(* IEC 61131-3 sources: mect_apps/TPAC1008_02_AF/Octopus_Prey/plc, 2 files *)

(* ---- Crosstable.gvl ---- *)
VAR_GLOBAL
	STATUS AT %QW0.772:UINT;
	RTU_HEARTBEAT AT %IW0.800:UINT;
	RTU_RTU_WR AT %QX0.804.0:BOOL;
	RTU_RTU_RD AT %IX0.808.0:BOOL;
	TEST_COMMAND AT %IW0.15896:UINT;
	TST_DigIn_1 AT %IX0.15900.0:BOOL;
	TST_DigIn_2 AT %IX0.15904.0:BOOL;
	TST_DigIn_3 AT %IX0.15908.0:BOOL;
	TST_DigIn_4 AT %IX0.15912.0:BOOL;
	TST_DigIn_5 AT %IX0.15916.0:BOOL;
	TST_DigIn_6 AT %IX0.15920.0:BOOL;
	TST_DigIn_7 AT %IX0.15924.0:BOOL;
	TST_DigIn_8 AT %IX0.15928.0:BOOL;
	TST_DigIn_9 AT %IX0.15932.0:BOOL;
	TST_DigIn_10 AT %IX0.15936.0:BOOL;
	TST_DigIn_11 AT %IX0.15940.0:BOOL;
	TST_DigIn_12 AT %IX0.15944.0:BOOL;
	TST_DigIn_13 AT %IX0.15948.0:BOOL;
	TST_DigIn_14 AT %IX0.15952.0:BOOL;
	TST_DigIn_15 AT %IX0.15956.0:BOOL;
	TST_DigIn_16 AT %IX0.15960.0:BOOL;
	VAL_DigIn_1 AT %IX0.15964.0:BOOL;
	VAL_DigIn_2 AT %IX0.15968.0:BOOL;
	VAL_DigIn_3 AT %IX0.15972.0:BOOL;
	VAL_DigIn_4 AT %IX0.15976.0:BOOL;
	VAL_DigIn_5 AT %IX0.15980.0:BOOL;
	VAL_DigIn_6 AT %IX0.15984.0:BOOL;
	VAL_DigIn_7 AT %IX0.15988.0:BOOL;
	VAL_DigIn_8 AT %IX0.15992.0:BOOL;
	VAL_DigIn_9 AT %IX0.15996.0:BOOL;
	VAL_DigIn_10 AT %IX0.16000.0:BOOL;
	VAL_DigIn_11 AT %IX0.16004.0:BOOL;
	VAL_DigIn_12 AT %IX0.16008.0:BOOL;
	VAL_DigIn_13 AT %IX0.16012.0:BOOL;
	VAL_DigIn_14 AT %IX0.16016.0:BOOL;
	VAL_DigIn_15 AT %IX0.16020.0:BOOL;
	VAL_DigIn_16 AT %IX0.16024.0:BOOL;
	RES_DigIn_1 AT %QX0.16028.0:BOOL;
	RES_DigIn_2 AT %QX0.16032.0:BOOL;
	RES_DigIn_3 AT %QX0.16036.0:BOOL;
	RES_DigIn_4 AT %QX0.16040.0:BOOL;
	RES_DigIn_5 AT %QX0.16044.0:BOOL;
	RES_DigIn_6 AT %QX0.16048.0:BOOL;
	RES_DigIn_7 AT %QX0.16052.0:BOOL;
	RES_DigIn_8 AT %QX0.16056.0:BOOL;
	RES_DigIn_9 AT %QX0.16060.0:BOOL;
	RES_DigIn_10 AT %QX0.16064.0:BOOL;
	RES_DigIn_11 AT %QX0.16068.0:BOOL;
	RES_DigIn_12 AT %QX0.16072.0:BOOL;
	RES_DigIn_13 AT %QX0.16076.0:BOOL;
	RES_DigIn_14 AT %QX0.16080.0:BOOL;
	RES_DigIn_15 AT %QX0.16084.0:BOOL;
	RES_DigIn_16 AT %QX0.16088.0:BOOL;
	TST_DigOut_1 AT %IX0.16092.0:BOOL;
	TST_DigOut_2 AT %IX0.16096.0:BOOL;
	TST_DigOut_3 AT %IX0.16100.0:BOOL;
	TST_DigOut_4 AT %IX0.16104.0:BOOL;
	TST_DigOut_5 AT %IX0.16108.0:BOOL;
	TST_DigOut_6 AT %IX0.16112.0:BOOL;
	TST_DigOut_7 AT %IX0.16116.0:BOOL;
	TST_DigOut_8 AT %IX0.16120.0:BOOL;
	TST_DigOut_9 AT %IX0.16124.0:BOOL;
	TST_DigOut_10 AT %IX0.16128.0:BOOL;
	TST_DigOut_11 AT %IX0.16132.0:BOOL;
	TST_DigOut_12 AT %IX0.16136.0:BOOL;
	TST_DigOut_13 AT %IX0.16140.0:BOOL;
	TST_DigOut_14 AT %IX0.16144.0:BOOL;
	TST_DigOut_15 AT %IX0.16148.0:BOOL;
	TST_DigOut_16 AT %IX0.16152.0:BOOL;
	VAL_DigOut_1 AT %IX0.16156.0:BOOL;
	VAL_DigOut_2 AT %IX0.16160.0:BOOL;
	VAL_DigOut_3 AT %IX0.16164.0:BOOL;
	VAL_DigOut_4 AT %IX0.16168.0:BOOL;
	VAL_DigOut_5 AT %IX0.16172.0:BOOL;
	VAL_DigOut_6 AT %IX0.16176.0:BOOL;
	VAL_DigOut_7 AT %IX0.16180.0:BOOL;
	VAL_DigOut_8 AT %IX0.16184.0:BOOL;
	VAL_DigOut_9 AT %IX0.16188.0:BOOL;
	VAL_DigOut_10 AT %IX0.16192.0:BOOL;
	VAL_DigOut_11 AT %IX0.16196.0:BOOL;
	VAL_DigOut_12 AT %IX0.16200.0:BOOL;
	VAL_DigOut_13 AT %IX0.16204.0:BOOL;
	VAL_DigOut_14 AT %IX0.16208.0:BOOL;
	VAL_DigOut_15 AT %IX0.16212.0:BOOL;
	VAL_DigOut_16 AT %IX0.16216.0:BOOL;
	TST_AnIn_1 AT %IX0.16220.0:BOOL;
	TST_AnIn_2 AT %IX0.16224.0:BOOL;
	TST_AnIn_3 AT %IX0.16228.0:BOOL;
	TST_AnIn_4 AT %IX0.16232.0:BOOL;
	TST_AnIn_5 AT %IX0.16236.0:BOOL;
	TST_AnIn_6 AT %IX0.16240.0:BOOL;
	TST_AnIn_7 AT %IX0.16244.0:BOOL;
	TST_AnIn_8 AT %IX0.16248.0:BOOL;
	TST_AnIn_9 AT %IX0.16252.0:BOOL;
	TST_AnIn_10 AT %IX0.16256.0:BOOL;
	TST_AnIn_11 AT %IX0.16260.0:BOOL;
	TST_AnIn_12 AT %IX0.16264.0:BOOL;
	VAL_AnIn_1 AT %IW0.16268:INT;
	VAL_AnIn_2 AT %IW0.16272:INT;
	VAL_AnIn_3 AT %IW0.16276:INT;
	VAL_AnIn_4 AT %IW0.16280:INT;
	VAL_AnIn_5 AT %IW0.16284:INT;
	VAL_AnIn_6 AT %IW0.16288:INT;
	VAL_AnIn_7 AT %IW0.16292:INT;
	VAL_AnIn_8 AT %IW0.16296:INT;
	VAL_AnIn_9 AT %IW0.16300:INT;
	VAL_AnIn_10 AT %IW0.16304:INT;
	VAL_AnIn_11 AT %IW0.16308:INT;
	VAL_AnIn_12 AT %IW0.16312:INT;
	VAL_AnInConf_1 AT %IW0.16316:UINT;
	VAL_AnInConf_2 AT %IW0.16320:UINT;
	VAL_AnInConf_3 AT %IW0.16324:UINT;
	VAL_AnInConf_4 AT %IW0.16328:UINT;
	VAL_AnInConf_5 AT %IW0.16332:UINT;
	VAL_AnInConf_6 AT %IW0.16336:UINT;
	VAL_AnInConf_7 AT %IW0.16340:UINT;
	VAL_AnInConf_8 AT %IW0.16344:UINT;
	VAL_AnInConf_9 AT %IW0.16348:UINT;
	VAL_AnInConf_10 AT %IW0.16352:UINT;
	VAL_AnInConf_11 AT %IW0.16356:UINT;
	VAL_AnInConf_12 AT %IW0.16360:UINT;
	VAL_AnInFltr_1 AT %IW0.16364:UINT;
	VAL_AnInFltr_2 AT %IW0.16368:UINT;
	VAL_AnInFltr_3 AT %IW0.16372:UINT;
	VAL_AnInFltr_4 AT %IW0.16376:UINT;
	VAL_AnInFltr_5 AT %IW0.16380:UINT;
	VAL_AnInFltr_6 AT %IW0.16384:UINT;
	VAL_AnInFltr_7 AT %IW0.16388:UINT;
	VAL_AnInFltr_8 AT %IW0.16392:UINT;
	VAL_AnInFltr_9 AT %IW0.16396:UINT;
	VAL_AnInFltr_10 AT %IW0.16400:UINT;
	VAL_AnInFltr_11 AT %IW0.16404:UINT;
	VAL_AnInFltr_12 AT %IW0.16408:UINT;
	RES_AnIn_1 AT %QW0.16412:INT;
	RES_AnIn_2 AT %QW0.16416:INT;
	RES_AnIn_3 AT %QW0.16420:INT;
	RES_AnIn_4 AT %QW0.16424:INT;
	RES_AnIn_5 AT %QW0.16428:INT;
	RES_AnIn_6 AT %QW0.16432:INT;
	RES_AnIn_7 AT %QW0.16436:INT;
	RES_AnIn_8 AT %QW0.16440:INT;
	RES_AnIn_9 AT %QW0.16444:INT;
	RES_AnIn_10 AT %QW0.16448:INT;
	RES_AnIn_11 AT %QW0.16452:INT;
	RES_AnIn_12 AT %QW0.16456:INT;
	RES_AnInStts_1 AT %QW0.16460:INT;
	RES_AnInStts_2 AT %QW0.16464:INT;
	RES_AnInStts_3 AT %QW0.16468:INT;
	RES_AnInStts_4 AT %QW0.16472:INT;
	RES_AnInStts_5 AT %QW0.16476:INT;
	RES_AnInStts_6 AT %QW0.16480:INT;
	RES_AnInStts_7 AT %QW0.16484:INT;
	RES_AnInStts_8 AT %QW0.16488:INT;
	RES_AnInStts_9 AT %QW0.16492:INT;
	RES_AnInStts_10 AT %QW0.16496:INT;
	RES_AnInStts_11 AT %QW0.16500:INT;
	RES_AnInStts_12 AT %QW0.16504:INT;
	TST_AnOut_1 AT %IX0.16508.0:BOOL;
	TST_AnOut_2 AT %IX0.16512.0:BOOL;
	TST_AnOut_3 AT %IX0.16516.0:BOOL;
	TST_AnOut_4 AT %IX0.16520.0:BOOL;
	VAL_AnOut_1 AT %IW0.16524:INT;
	VAL_AnOut_2 AT %IW0.16528:INT;
	VAL_AnOut_3 AT %IW0.16532:INT;
	VAL_AnOut_4 AT %IW0.16536:INT;
	VAL_AnOutConf_1 AT %IW0.16540:UINT;
	VAL_AnOutConf_2 AT %IW0.16544:UINT;
	VAL_AnOutConf_3 AT %IW0.16548:UINT;
	VAL_AnOutConf_4 AT %IW0.16552:UINT;
	RES_AnOutStts_1 AT %QW0.16556:INT;
	RES_AnOutStts_2 AT %QW0.16560:INT;
	RES_AnOutStts_3 AT %QW0.16564:INT;
	RES_AnOutStts_4 AT %QW0.16568:INT;
	TST_Tamb AT %IX0.16572.0:BOOL;
	TST_RPM AT %IX0.16576.0:BOOL;
	TST_FWrevision AT %IX0.16580.0:BOOL;
	TST_HWconfig AT %IX0.16584.0:BOOL;
	VAL_Tamb AT %IW0.16588:INT;
	VAL_RPM AT %IW0.16592:UINT;
	VAL_FWrevision AT %IW0.16596:UINT;
	VAL_HWconfig AT %IW0.16600:UINT;
	RES_Tamb AT %QW0.16604:INT;
	RES_RPM AT %QW0.16608:UINT;
	RES_FWrevision AT %QW0.16612:UINT;
	RES_HWconfig AT %QW0.16616:UINT;
	TST_RTUS_WR AT %IX0.16620.0:BOOL;
	TST_RTUS_RD AT %IX0.16624.0:BOOL;
	TST_RTU1_WR AT %IX0.16628.0:BOOL;
	TST_RTU1_RD AT %IX0.16632.0:BOOL;
	TST_RTU3_WR AT %IX0.16636.0:BOOL;
	TST_RTU3_RD AT %IX0.16640.0:BOOL;
	TST_CAN1_WR AT %IX0.16644.0:BOOL;
	TST_CAN1_RD AT %IX0.16648.0:BOOL;
	VAL_RTUS_WR AT %IX0.16652.0:BOOL;
	VAL_RTUS_RD AT %IX0.16656.0:BOOL;
	VAL_RTU1_WR AT %IX0.16660.0:BOOL;
	VAL_RTU1_RD AT %IX0.16664.0:BOOL;
	VAL_RTU3_WR AT %IX0.16668.0:BOOL;
	VAL_RTU3_RD AT %IX0.16672.0:BOOL;
	VAL_CAN1_WR AT %IX0.16676.0:BOOL;
	VAL_CAN1_RD AT %IX0.16680.0:BOOL;
	RES_RTUS_WR AT %QX0.16684.0:BOOL;
	RES_RTUS_RD AT %QX0.16688.0:BOOL;
	RES_RTU1_WR AT %QX0.16692.0:BOOL;
	RES_RTU1_RD AT %QX0.16696.0:BOOL;
	RES_RTU3_WR AT %QX0.16700.0:BOOL;
	RES_RTU3_RD AT %QX0.16704.0:BOOL;
	RES_CAN1_WR AT %QX0.16708.0:BOOL;
	RES_CAN1_RD AT %QX0.16712.0:BOOL;
	TEST_STATUS AT %QW0.16716:UINT;
	RTU0_TYPE_PORT AT %ID0.20000:UDINT;
	RTU0_BAUDRATE AT %ID0.20004:UDINT;
	RTU0_STATUS AT %ID0.20008:UDINT;
	RTU0_READS AT %ID0.20012:UDINT;
	RTU0_WRITES AT %ID0.20016:UDINT;
	RTU0_TIMEOUTS AT %ID0.20020:UDINT;
	RTU0_COMM_ERRORS AT %ID0.20024:UDINT;
	RTU0_LAST_ERROR AT %ID0.20028:UDINT;
	RTU0_WRITE_QUEUE AT %ID0.20032:UDINT;
	RTU0_BUS_LOAD AT %ID0.20036:UDINT;
	RTU1_TYPE_PORT AT %ID0.20040:UDINT;
	RTU1_BAUDRATE AT %ID0.20044:UDINT;
	RTU1_STATUS AT %ID0.20048:UDINT;
	RTU1_READS AT %ID0.20052:UDINT;
	RTU1_WRITES AT %ID0.20056:UDINT;
	RTU1_TIMEOUTS AT %ID0.20060:UDINT;
	RTU1_COMM_ERRORS AT %ID0.20064:UDINT;
	RTU1_LAST_ERROR AT %ID0.20068:UDINT;
	RTU1_WRITE_QUEUE AT %ID0.20072:UDINT;
	RTU1_BUS_LOAD AT %ID0.20076:UDINT;
	RTU3_TYPE_PORT AT %ID0.20080:UDINT;
	RTU3_BAUDRATE AT %ID0.20084:UDINT;
	RTU3_STATUS AT %ID0.20088:UDINT;
	RTU3_READS AT %ID0.20092:UDINT;
	RTU3_WRITES AT %ID0.20096:UDINT;
	RTU3_TIMEOUTS AT %ID0.20100:UDINT;
	RTU3_COMM_ERRORS AT %ID0.20104:UDINT;
	RTU3_LAST_ERROR AT %ID0.20108:UDINT;
	RTU3_WRITE_QUEUE AT %ID0.20112:UDINT;
	RTU3_BUS_LOAD AT %ID0.20116:UDINT;
	CAN0_TYPE_PORT AT %ID0.20120:UDINT;
	CAN0_BAUDRATE AT %ID0.20124:UDINT;
	CAN0_STATUS AT %ID0.20128:UDINT;
	CAN0_READS AT %ID0.20132:UDINT;
	CAN0_WRITES AT %ID0.20136:UDINT;
	CAN0_TIMEOUTS AT %ID0.20140:UDINT;
	CAN0_COMM_ERRORS AT %ID0.20144:UDINT;
	CAN0_LAST_ERROR AT %ID0.20148:UDINT;
	CAN0_WRITE_QUEUE AT %ID0.20152:UDINT;
	CAN0_BUS_LOAD AT %ID0.20156:UDINT;
	CAN1_TYPE_PORT AT %ID0.20160:UDINT;
	CAN1_BAUDRATE AT %ID0.20164:UDINT;
	CAN1_STATUS AT %ID0.20168:UDINT;
	CAN1_READS AT %ID0.20172:UDINT;
	CAN1_WRITES AT %ID0.20176:UDINT;
	CAN1_TIMEOUTS AT %ID0.20180:UDINT;
	CAN1_COMM_ERRORS AT %ID0.20184:UDINT;
	CAN1_LAST_ERROR AT %ID0.20188:UDINT;
	CAN1_WRITE_QUEUE AT %ID0.20192:UDINT;
	CAN1_BUS_LOAD AT %ID0.20196:UDINT;
	TCPS_TYPE_PORT AT %ID0.20200:UDINT;
	TCPS_IP_ADDRESS AT %ID0.20204:UDINT;
	TCPS_STATUS AT %ID0.20208:UDINT;
	TCPS_READS AT %ID0.20212:UDINT;
	TCPS_WRITES AT %ID0.20216:UDINT;
	TCPS_TIMEOUTS AT %ID0.20220:UDINT;
	TCPS_COMM_ERRORS AT %ID0.20224:UDINT;
	TCPS_LAST_ERROR AT %ID0.20228:UDINT;
	TCPS_WRITE_QUEUE AT %ID0.20232:UDINT;
	TCPS_BUS_LOAD AT %ID0.20236:UDINT;
	TCP0_TYPE_PORT AT %ID0.20240:UDINT;
	TCP0_IP_ADDRESS AT %ID0.20244:UDINT;
	TCP0_STATUS AT %ID0.20248:UDINT;
	TCP0_READS AT %ID0.20252:UDINT;
	TCP0_WRITES AT %ID0.20256:UDINT;
	TCP0_TIMEOUTS AT %ID0.20260:UDINT;
	TCP0_COMM_ERRORS AT %ID0.20264:UDINT;
	TCP0_LAST_ERROR AT %ID0.20268:UDINT;
	TCP0_WRITE_QUEUE AT %ID0.20272:UDINT;
	TCP0_BUS_LOAD AT %ID0.20276:UDINT;
	TCP1_TYPE_PORT AT %ID0.20280:UDINT;
	TCP1_IP_ADDRESS AT %ID0.20284:UDINT;
	TCP1_STATUS AT %ID0.20288:UDINT;
	TCP1_READS AT %ID0.20292:UDINT;
	TCP1_WRITES AT %ID0.20296:UDINT;
	TCP1_TIMEOUTS AT %ID0.20300:UDINT;
	TCP1_COMM_ERRORS AT %ID0.20304:UDINT;
	TCP1_LAST_ERROR AT %ID0.20308:UDINT;
	TCP1_WRITE_QUEUE AT %ID0.20312:UDINT;
	TCP1_BUS_LOAD AT %ID0.20316:UDINT;
	TCP2_TYPE_PORT AT %ID0.20320:UDINT;
	TCP2_IP_ADDRESS AT %ID0.20324:UDINT;
	TCP2_STATUS AT %ID0.20328:UDINT;
	TCP2_READS AT %ID0.20332:UDINT;
	TCP2_WRITES AT %ID0.20336:UDINT;
	TCP2_TIMEOUTS AT %ID0.20340:UDINT;
	TCP2_COMM_ERRORS AT %ID0.20344:UDINT;
	TCP2_LAST_ERROR AT %ID0.20348:UDINT;
	TCP2_WRITE_QUEUE AT %ID0.20352:UDINT;
	TCP2_BUS_LOAD AT %ID0.20356:UDINT;
	TCP3_TYPE_PORT AT %ID0.20360:UDINT;
	TCP3_IP_ADDRESS AT %ID0.20364:UDINT;
	TCP3_STATUS AT %ID0.20368:UDINT;
	TCP3_READS AT %ID0.20372:UDINT;
	TCP3_WRITES AT %ID0.20376:UDINT;
	TCP3_TIMEOUTS AT %ID0.20380:UDINT;
	TCP3_COMM_ERRORS AT %ID0.20384:UDINT;
	TCP3_LAST_ERROR AT %ID0.20388:UDINT;
	TCP3_WRITE_QUEUE AT %ID0.20392:UDINT;
	TCP3_BUS_LOAD AT %ID0.20396:UDINT;
	TCP4_TYPE_PORT AT %ID0.20400:UDINT;
	TCP4_IP_ADDRESS AT %ID0.20404:UDINT;
	TCP4_STATUS AT %ID0.20408:UDINT;
	TCP4_READS AT %ID0.20412:UDINT;
	TCP4_WRITES AT %ID0.20416:UDINT;
	TCP4_TIMEOUTS AT %ID0.20420:UDINT;
	TCP4_COMM_ERRORS AT %ID0.20424:UDINT;
	TCP4_LAST_ERROR AT %ID0.20428:UDINT;
	TCP4_WRITE_QUEUE AT %ID0.20432:UDINT;
	TCP4_BUS_LOAD AT %ID0.20436:UDINT;
	TCP5_TYPE_PORT AT %ID0.20440:UDINT;
	TCP5_IP_ADDRESS AT %ID0.20444:UDINT;
	TCP5_STATUS AT %ID0.20448:UDINT;
	TCP5_READS AT %ID0.20452:UDINT;
	TCP5_WRITES AT %ID0.20456:UDINT;
	TCP5_TIMEOUTS AT %ID0.20460:UDINT;
	TCP5_COMM_ERRORS AT %ID0.20464:UDINT;
	TCP5_LAST_ERROR AT %ID0.20468:UDINT;
	TCP5_WRITE_QUEUE AT %ID0.20472:UDINT;
	TCP5_BUS_LOAD AT %ID0.20476:UDINT;
	TCP6_TYPE_PORT AT %ID0.20480:UDINT;
	TCP6_IP_ADDRESS AT %ID0.20484:UDINT;
	TCP6_STATUS AT %ID0.20488:UDINT;
	TCP6_READS AT %ID0.20492:UDINT;
	TCP6_WRITES AT %ID0.20496:UDINT;
	TCP6_TIMEOUTS AT %ID0.20500:UDINT;
	TCP6_COMM_ERRORS AT %ID0.20504:UDINT;
	TCP6_LAST_ERROR AT %ID0.20508:UDINT;
	TCP6_WRITE_QUEUE AT %ID0.20512:UDINT;
	TCP6_BUS_LOAD AT %ID0.20516:UDINT;
	TCP7_TYPE_PORT AT %ID0.20520:UDINT;
	TCP7_IP_ADDRESS AT %ID0.20524:UDINT;
	TCP7_STATUS AT %ID0.20528:UDINT;
	TCP7_READS AT %ID0.20532:UDINT;
	TCP7_WRITES AT %ID0.20536:UDINT;
	TCP7_TIMEOUTS AT %ID0.20540:UDINT;
	TCP7_COMM_ERRORS AT %ID0.20544:UDINT;
	TCP7_LAST_ERROR AT %ID0.20548:UDINT;
	TCP7_WRITE_QUEUE AT %ID0.20552:UDINT;
	TCP7_BUS_LOAD AT %ID0.20556:UDINT;
	TCP8_TYPE_PORT AT %ID0.20560:UDINT;
	TCP8_IP_ADDRESS AT %ID0.20564:UDINT;
	TCP8_STATUS AT %ID0.20568:UDINT;
	TCP8_READS AT %ID0.20572:UDINT;
	TCP8_WRITES AT %ID0.20576:UDINT;
	TCP8_TIMEOUTS AT %ID0.20580:UDINT;
	TCP8_COMM_ERRORS AT %ID0.20584:UDINT;
	TCP8_LAST_ERROR AT %ID0.20588:UDINT;
	TCP8_WRITE_QUEUE AT %ID0.20592:UDINT;
	TCP8_BUS_LOAD AT %ID0.20596:UDINT;
	TCP9_TYPE_PORT AT %ID0.20600:UDINT;
	TCP9_IP_ADDRESS AT %ID0.20604:UDINT;
	TCP9_STATUS AT %ID0.20608:UDINT;
	TCP9_READS AT %ID0.20612:UDINT;
	TCP9_WRITES AT %ID0.20616:UDINT;
	TCP9_TIMEOUTS AT %ID0.20620:UDINT;
	TCP9_COMM_ERRORS AT %ID0.20624:UDINT;
	TCP9_LAST_ERROR AT %ID0.20628:UDINT;
	TCP9_WRITE_QUEUE AT %ID0.20632:UDINT;
	TCP9_BUS_LOAD AT %ID0.20636:UDINT;
	NODE_01_DEV_NODE AT %ID0.20688:UDINT;
	NODE_01_STATUS AT %ID0.20692:UDINT;
	NODE_02_DEV_NODE AT %ID0.20696:UDINT;
	NODE_02_STATUS AT %ID0.20700:UDINT;
	NODE_03_DEV_NODE AT %ID0.20704:UDINT;
	NODE_03_STATUS AT %ID0.20708:UDINT;
	NODE_04_DEV_NODE AT %ID0.20712:UDINT;
	NODE_04_STATUS AT %ID0.20716:UDINT;
	NODE_05_DEV_NODE AT %ID0.20720:UDINT;
	NODE_05_STATUS AT %ID0.20724:UDINT;
	NODE_06_DEV_NODE AT %ID0.20728:UDINT;
	NODE_06_STATUS AT %ID0.20732:UDINT;
	NODE_07_DEV_NODE AT %ID0.20736:UDINT;
	NODE_07_STATUS AT %ID0.20740:UDINT;
	NODE_08_DEV_NODE AT %ID0.20744:UDINT;
	NODE_08_STATUS AT %ID0.20748:UDINT;
	NODE_09_DEV_NODE AT %ID0.20752:UDINT;
	NODE_09_STATUS AT %ID0.20756:UDINT;
	NODE_10_DEV_NODE AT %ID0.20760:UDINT;
	NODE_10_STATUS AT %ID0.20764:UDINT;
	NODE_11_DEV_NODE AT %ID0.20768:UDINT;
	NODE_11_STATUS AT %ID0.20772:UDINT;
	NODE_12_DEV_NODE AT %ID0.20776:UDINT;
	NODE_12_STATUS AT %ID0.20780:UDINT;
	NODE_13_DEV_NODE AT %ID0.20784:UDINT;
	NODE_13_STATUS AT %ID0.20788:UDINT;
	NODE_14_DEV_NODE AT %ID0.20792:UDINT;
	NODE_14_STATUS AT %ID0.20796:UDINT;
	NODE_15_DEV_NODE AT %ID0.20800:UDINT;
	NODE_15_STATUS AT %ID0.20804:UDINT;
	NODE_16_DEV_NODE AT %ID0.20808:UDINT;
	NODE_16_STATUS AT %ID0.20812:UDINT;
	PLC_DigIn_1 AT %IX0.21200.0:BOOL;	(* Digital input 1 value *)
	PLC_DigIn_2 AT %IX0.21204.0:BOOL;	(* Digital input 2 value *)
	PLC_DigIn_3 AT %IX0.21208.0:BOOL;	(* Digital input 3 value *)
	PLC_DigIn_4 AT %IX0.21212.0:BOOL;	(* Digital input 4 value *)
	PLC_DigIn_5 AT %IX0.21216.0:BOOL;	(* Digital input 5 value *)
	PLC_DigIn_6 AT %IX0.21220.0:BOOL;	(* Digital input 6 value *)
	PLC_DigIn_7 AT %IX0.21224.0:BOOL;	(* Digital input 7 value *)
	PLC_DigIn_8 AT %IX0.21228.0:BOOL;	(* Digital input 8 value *)
	PLC_Reserved_1 AT %IX0.21232.0:BOOL;	(* Reserved *)
	PLC_DigOut_1 AT %QX0.21236.0:BOOL;	(* Digital output 1 value *)
	PLC_DigOut_2 AT %QX0.21240.0:BOOL;	(* Digital output 2 value *)
	PLC_DigOut_3 AT %QX0.21244.0:BOOL;	(* Digital output 3 value *)
	PLC_DigOut_4 AT %QX0.21248.0:BOOL;	(* Digital output 4 value *)
	PLC_DigOut_5 AT %QX0.21252.0:BOOL;	(* Digital output 5 value *)
	PLC_DigOut_6 AT %QX0.21256.0:BOOL;	(* Digital output 6 value *)
	PLC_DigOut_7 AT %QX0.21260.0:BOOL;	(* Digital output 7 value *)
	PLC_DigOut_8 AT %QX0.21264.0:BOOL;	(* Digital output 8 value *)
	PLC_DigOut_9 AT %QX0.21268.0:BOOL;	(* Digital output 9 value *)
	PLC_DigOut_10 AT %QX0.21272.0:BOOL;	(* Digital output 10 value *)
	PLC_DigOut_11 AT %QX0.21276.0:BOOL;	(* Digital output 11 value *)
	PLC_DigOut_12 AT %QX0.21280.0:BOOL;	(* Digital output 12 value *)
	PLC_Hwconf AT %IW0.21284:UINT;	(* Hardware configuration *)
	PLC_Revisione AT %IW0.21288:UINT;	(* Firmware version *)
	PLC_StatusReg AT %IW0.21292:UINT;	(* In - Out board status *)
	PLC_Heartbeat AT %IW0.21296:UINT;	(* In - Out board function check *)
	PLC_AnIn_1 AT %IW0.21300:INT;	(* Analog input 1 value *)
	PLC_AnIn_2 AT %IW0.21304:INT;	(* Analog input 2 value *)
	PLC_AnIn_3 AT %IW0.21308:INT;	(* Analog input 3 value *)
	PLC_AnIn_4 AT %IW0.21312:INT;	(* Analog input 4 value *)
	PLC_EncoderCo_Lo AT %IW0.21316:UINT;	(* Encoder reading (LOW) *)
	PLC_EncoderCo_Hi AT %IW0.21320:UINT;	(* Encoder reading (HIGH) *)
	PLC_CaptureT1_Lo AT %IW0.21324:UINT;	(* Time between 2 input edges (LOW) *)
	PLC_CaptureT1_Hi AT %IW0.21328:UINT;	(* Time between 2 input edges (HIGH) *)
	PLC_CaptureT2_Lo AT %IW0.21332:UINT;	(* Time between 2 input edges (LOW) *)
	PLC_CaptureT2_Hi AT %IW0.21336:UINT;	(* Time between 2 input edges (HIGH) *)
	PLC_RPM AT %IW0.21340:UINT;	(* RPM input *)
	PLC_Tamb AT %IW0.21344:INT;	(* Cold junction compensation value *)
	PLC_EnableEnc AT %QW0.21348:UINT;	(* Encoder - counter enable *)
	PLC_ResetCount AT %QW0.21352:UINT;	(* Encoder reset *)
	PLC_AnInConf_1 AT %QW0.21356:UINT;	(* Analog input 1 configuration *)
	PLC_AnInConf_2 AT %QW0.21360:UINT;	(* Analog input 2 configuration *)
	PLC_AnInConf_3 AT %QW0.21364:UINT;	(* Analog input 3 configuration *)
	PLC_AnInConf_4 AT %QW0.21368:UINT;	(* Analog input 4 configuration *)
	PLC_AnOutConf_1 AT %QW0.21372:UINT;	(* Analog output 1 configuration *)
	PLC_AnOutConf_2 AT %QW0.21376:UINT;	(* Analog output 2 configuration *)
	PLC_AnOutConf_3 AT %QW0.21380:UINT;	(* Analog output 3 configuration *)
	PLC_AnOutConf_4 AT %QW0.21384:UINT;	(* Analog output 4 configuration *)
	PLC_AnOut_1 AT %QW0.21388:INT;	(* Analog output 1 value *)
	PLC_AnOut_2 AT %QW0.21392:INT;	(* Analog output 2 value *)
	PLC_AnOut_3 AT %QW0.21396:INT;	(* Analog output 3 value *)
	PLC_AnOut_4 AT %QW0.21400:INT;	(* Analog output 4 value *)
	PLC_FiltAnIn_1 AT %QW0.21404:UINT;	(* Analog input 1 filter *)
	PLC_FiltAnIn_2 AT %QW0.21408:UINT;	(* Analog input 2 filter *)
	PLC_FiltAnIn_3 AT %QW0.21412:UINT;	(* Analog input 3 filter *)
	PLC_FiltAnIn_4 AT %QW0.21416:UINT;	(* Analog input 4 filter *)
	CH0_NETRUN AT %IX0.21428.0:BOOL;	(* Active channel *)
	CH0_NETGOOD AT %IX0.21432.0:BOOL;	(* Channel configuration *)
	CH0_NETERR AT %ID0.21436:UDINT;	(* Bus status *)
	CH0_NETRST AT %QX0.21440.0:BOOL;	(* Bus reset *)
	CH0_NETDIS AT %QX0.21444.0:BOOL;	(* Disable the bus *)
	CH0_01_NODERUN AT %IX0.21448.0:BOOL;	(* In Out board - active channel *)
	CH0_01_NODEGOOD AT %IX0.21452.0:BOOL;	(* In Out board - channel configuration *)
	CH0_01_NODEERR AT %ID0.21456:UDINT;	(* In Out board - bus status *)
	CH0_01_NODERST AT %QX0.21460.0:BOOL;	(* In Out board - bus reset *)
	CH0_01_NODEDIS AT %QX0.21464.0:BOOL;	(* In Out board - disable the bus *)
	PLC_time AT %ID0.21560:REAL;	(* Seconds since boot (reset each 24h) *)
	PLC_timeMin AT %ID0.21564:REAL;	(* 10 seconds window start *)
	PLC_timeMax AT %ID0.21568:REAL;	(* 10 seconds window stop *)
	PLC_timeWin AT %QD0.21572:REAL;	(* Graph display window *)
	PLC_Version AT %IW0.21576:UINT;	(* Run Time version *)
	PLC_EngineStatus AT %IW0.21580:UINT;	(* PLC status *)
	PLC_ResetValues AT %QX0.21584.0:BOOL;	(* Diagnostic variables reset *)
	PLC_buzzerOn AT %QX0.21588.0:BOOL;	(* Buzzer sound (enable = 1 disable = 0) *)
	PLC_PLC_Version AT %QW0.21592:UINT;	(* PLC application version *)
	PLC_HMI_Version AT %QW0.21596:UINT;	(* HMI application version *)
	PLC_Year AT %IW0.21640:UINT;	(* Currently year *)
	PLC_Month AT %IW0.21644:UINT;	(* Currently month *)
	PLC_Day AT %IW0.21648:UINT;	(* Currently day *)
	PLC_Hours AT %IW0.21652:UINT;	(* Currently hour *)
	PLC_Minutes AT %IW0.21656:UINT;	(* Currently minutes *)
	PLC_Seconds AT %IW0.21660:UINT;	(* Currently seconds *)
	PLC_UPTIME_s AT %ID0.21664:UDINT;	(* Uptime in seconds (wraps in 136 years) *)
	PLC_UPTIME_cs AT %ID0.21668:UDINT;	(* Uptime in centiseconds = 10 ms (wraps in 497 days) *)
	PLC_WATCHDOGEN AT %QX0.21672.0:BOOL;	(* Enable Watchdog *)
	PLC_WATCHDOG_ms AT %QD0.21676:UDINT;	(* Reset Watchdog timer *)
	PLC_PRODUCT_ID AT %ID0.21680:UDINT;	(* TP/TPAC/TPLC Product ID (Hex) *)
	PLC_SERIAL_NUMBER AT %ID0.21684:UDINT;	(* TP/TPAC/TPLC Serial Number *)
	PLC_HMI_PAGE AT %QD0.21688:DINT;	(* HMI Page (page100=0x00000100) *)
	PLC_MS_VERSION AT %ID0.21692:UDINT;	(* Mect Suite Version installed on Target (0 if before 3.4.0) *)
	PLC_BEEP_VOLUME AT %QB0.21740:BYTE;	(* Beep volume (when buzzerOn) *)
	PLC_TOUCH_VOLUME AT %QB0.21744:BYTE;	(* Touch volume *)
	PLC_ALARM_VOLUME AT %QB0.21748:BYTE;	(* Alarm volume (when alarm) *)
	PLC_BUZZER AT %QD0.21752:UDINT;	(* Enable dynamic buzzer sound (0x44332211 up=0x11(%) on=0x22(cs) off=0x33(cs) rep=0x44(times)) *)
END_VAR

(* ---- Init.st ---- *)
(*[[
]]*)
PROGRAM Init
#import "Crosstable.gvl"

	PLC_AnInConf_1 := 2; (* 0..10V *)
	PLC_AnInConf_2 := 2; (* 0..10V *)
	PLC_AnInConf_3 := 2; (* 0..10V *)
	PLC_AnInConf_4 := 2; (* 0..10V *)

	PLC_AnOutConf_1 := 2; (* 0..10V *)
	PLC_AnOutConf_2 := 2; (* 0..10V *)

	TEST_STATUS := STATUS_LOCAL;

END_PROGRAM
